// Mitsubishi GX Works2 project: z18   PLC: Q02/Q02H

PROGRAM MAIN
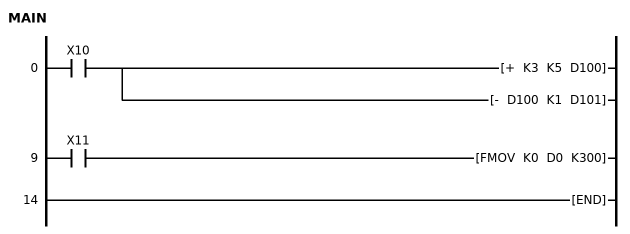
0     LD      X10
      +       K3 K5 D100
      -       D100 K1 D101
9     LD      X11
      FMOV    K0 D0 K300
14    END
END_PROGRAM
